(* IEC 61131-3 sources: Industry-PLC-LLM/data/PLCBEAD_repo/PLCBEAD_PLCEmbed-main/PLC-BEAD/Source/GEB/BYTE_TO_GRAY, 1 file *)

(* ---- BYTE_TO_GRAY.ST ---- *)
FUNCTION BYTE_TO_GRAY:BYTE
	VAR_INPUT
		IN :	BYTE;
	END_VAR

	BYTE_TO_GRAY := IN XOR SHR(IN,1);
END_FUNCTION

PROGRAM program0
  VAR
    LocalVar0 : BYTE;
    CEIL5_OUT : BYTE;
  END_VAR

  CEIL5_OUT := BYTE_TO_GRAY(LocalVar0);
END_PROGRAM
